// TIA Portal V19 export
TYPE "typeVfdInterface"
// stored: Access Published
   STRUCT
      general : "typeVfdGeneral";
      manual : "typeVfdManual";
      production : "typeVfdProduction";
      maintenance { S7_SetPoint := 'True'} : "typeVfdMaintenance";
   END_STRUCT;
END_TYPE
